(* PLC project C, V P 1 *)
(* stored: creationDateTime 2026-01-01T00:00:00 *)

PROGRAM Main
  VAR
    X : INT;
  END_VAR

X := X + 1;
END_PROGRAM
